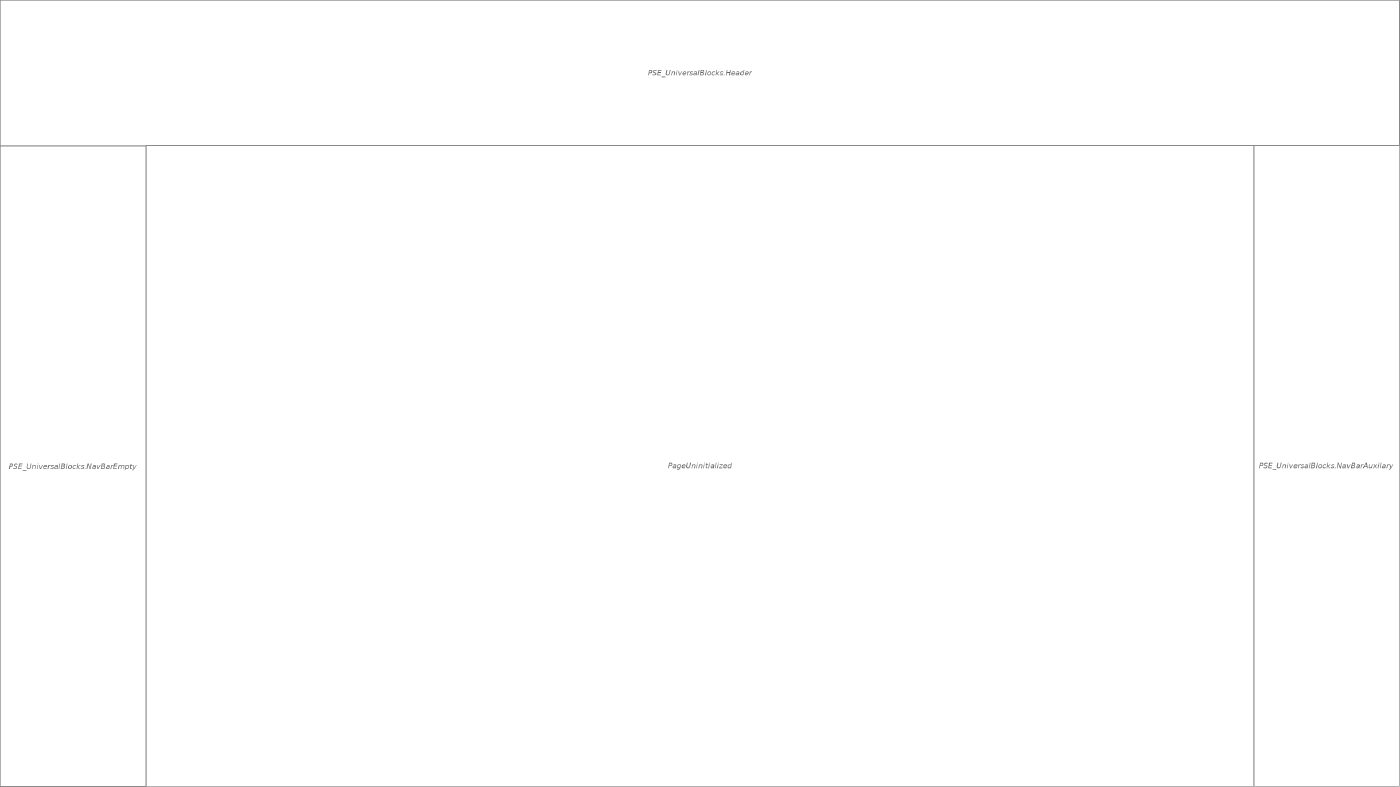
VISUALIZATION ShellMainVisu  // 1920x1080
    Frame (0,0 1920x200)
        shows PSE_UniversalBlocks.Header(sMachineName := PRG_VisuControl.fbVisuControl.sMachineName, sSoftwareVersion := PRG_VisuControl.fbVisuControl.sSoftwareVersion, eMachineState := PRG_MachineControl.fbMachineControler.State, sCurrentRecipe := PRG_VisuControl.fbVisuControl.sCurrentRecipe, sCurrentUser := PRG_VisuControl.fbVisuControl.sCurrentUser, iActiveCriticals := PRG_VisuControl.fbVisuControl.iActiveCriticals, iActvieErrors := PRG_VisuControl.fbVisuControl.iActvieErrors, iActiveWarrnings := PRG_VisuControl.fbVisuControl.iActiveWarrnings, sCurrentDate := PRG_VisuControl.fbVisuControl.sCurrentDate, sCurrentTime := PRG_VisuControl.fbVisuControl.sCurrentTime)
    Frame (0,200 200x880), frame switch variable: PRG_VisuControl.fbVisuControl.eCurrentNavigation
        shows PSE_UniversalBlocks.NavBarEmpty()
        shows PSE_UniversalBlocks.NavBarUninitialized(btnInitialize := PRG_VisuControl.fbVisuControl.btnInit)
        shows PSE_UniversalBlocks.NavBarInitializing(btnAbort := PRG_VisuControl.fbVisuControl.btnAbort)
        shows PSE_UniversalBlocks.NavBarAuto(btnStart := PRG_VisuControl.fbVisuControl.btnStart, btnStop := PRG_VisuControl.fbVisuControl.btnStop, btnManualMode := PRG_VisuControl.fbVisuControl.btnManual, btnAbort := PRG_VisuControl.fbVisuControl.btnAbort, btnReset := PRG_VisuControl.fbVisuControl.btnReset, bVisStart := PRG_VisuControl.fbVisuControl.bStartDisable, bVisStop := PRG_VisuControl.fbVisuControl.bStopDisable)
        shows PSE_UniversalBlocks.NavBarManual(btnAutoMode := PRG_VisuControl.fbVisuControl.btnAuto, btnCylinders := PRG_VisuControl.fbVisuControl.btnManualCylinder, btnMotors := PRG_VisuControl.fbVisuControl.btnManualAxis, btnSafety := PRG_VisuControl.fbVisuControl.btnManualSafety, btnInputs := PRG_VisuControl.fbVisuControl.btnManualInputs, btnOutputs := PRG_VisuControl.fbVisuControl.btnManualOutputs, btnOthers := PRG_VisuControl.fbVisuControl.btnManualOthers, btnAbort := PRG_VisuControl.fbVisuControl.btnAbort, btnRobots := PRG_VisuControl.fbVisuControl.btnManualRobots)
        shows PSE_UniversalBlocks.NavBarUtilities(btnBack := PRG_VisuControl.fbVisuControl.btnBack)
        shows PSE_UniversalBlocks.NavBarManual(btnAutoMode := PRG_Visu_Control.fbVisuControl.btnAuto, btnCylinders := PRG_Visu_Control.fbVisuControl.btnManualCylinder, btnMotors := PRG_Visu_Control.fbVisuControl.btnManualAxis, btnSafety := PRG_Visu_Control.fbVisuControl.btnManualSafety, btnInputs := PRG_Visu_Control.fbVisuControl.btnManualInputs, btnOutputs := PRG_Visu_Control.fbVisuControl.btnManualOutputs, btnOthers := PRG_Visu_Control.fbVisuControl.btnManualOthers, btnAbort := PRG_Visu_Control.fbVisuControl.btnAbort)
        shows PSE_UniversalBlocks.NavBarUtilities()
        shows PSE_UniversalBlocks.NavBarManual()
        shows PSE_UniversalBlocks.NavBarAuxilary(btnAlarms := PRG_Visu_Control.fbVisuControl.btnAlarms, btnRecipes := PRG_Visu_Control.fbVisuControl.btnRecipes, btnLights := PRG_Visu_Control.fbVisuControl.btnLights, sCloseHMIFileName := PRG_Visu_Control.fbVisuControl.sCloseHMIFileName, sCloseHMIParameters := PRG_Visu_Control.fbVisuControl.sCloseHMIParameters, bVisNotInit := PRG_Visu_Control.fbVisuControl.bVisNotInit, bVisHmiCLose := PRG_Visu_Control.fbVisuControl.bVisHmiClose, bVisLogIn := PRG_Visu_Control.fbVisuControl.bVisLogIn, bVisLogOut := PRG_Visu_Control.fbVisuControl.bVisLogOut)
        p2191133907: PRG_FB_Visu_Test.fbVisuControl.btnTest
        p3449907010: PRG_FB_Visu_Test.fbVisuControl.btnProcess
        p1834510317: PRG_FB_Visu_Test.fbVisuControl.btnTest
        p272088775: PRG_FB_Visu_Test.fbVisuControl.btnProcess
        p1969354770: PRG_FB_Visu_Test.fbVisuControl.btnAbort
        p1714963132: PRG_FB_Visu_Test.fbVisuControl.btnPushersScreenEntry
        p2303688632: PRG_FB_Visu_Test.fbVisuControl.btnStartAuto
        p3820184681: PRG_FB_Visu_Test.fbVisuControl.btnStop
        p1769496127: PRG_FB_Visu_Test.fbVisuControl.btnStepMode
        p2661042519: PRG_FB_Visu_Test.fbVisuControl.btnManual
        p976602031: PRG_VisuControl.fbVisuControl.btnBack
        p864465659: PRG_Visu_Control.fbVisuControl.ifUniversalMachineLink
        p1643820539: PRG_Visu_Control.fbVisuControl.btnStart
        p4004320302: PRG_Visu_Control.fbVisuControl.btnStop
        p3440189619: PRG_Visu_Control.fbVisuControl.btnManual
        p2317368076: PRG_Visu_Control.fbVisuControl.bVisStart
        p974511339: PRG_Visu_Control.fbVisuControl.bVisStop
        p3194361968: PRG_VisuControl.fbVisuControl.btnAuto
        p3852855334: PRG_VisuControl.fbVisuControl.btnManualCylinder
        p2703927093: PRG_VisuControl.fbVisuControl.btnManualAxis
        p1724788453: PRG_VisuControl.fbVisuControl.btnManualSafety
        p3478313700: PRG_VisuControl.fbVisuControl.btnManualInputs
        p985323216: PRG_VisuControl.fbVisuControl.btnManualOutputs
        p3968519516: PRG_VisuControl.fbVisuControl.btnManualOthers
        p3317205904: PRG_VisuControl.fbVisuControl.btnAbort
        p1887615166: PRG_VisuControl.fbVisuControl.btnManualRobots
    Frame (1719,199 200x880)
        shows PSE_UniversalBlocks.NavBarAuxilary(btnAlarms := PRG_VisuControl.fbVisuControl.btnAlarms, btnRecipes := PRG_VisuControl.fbVisuControl.btnRecipes, btnDoorLock := PRG_VisuControl.fbVisuControl.btnLights, btnLogIn := PRG_VisuControl.fbVisuControl.btnLogIn, btnLogOut := PRG_VisuControl.fbVisuControl.btnLogOut, btnHmiClose := PRG_VisuControl.fbVisuControl.btnHmiClose, sCloseHMIFileName := PRG_VisuControl.fbVisuControl.sCloseHMIFileName, sCloseHMIParameters := PRG_VisuControl.fbVisuControl.sCloseHMIParameters, bVisNotInit := PRG_VisuControl.fbVisuControl.bVisNotInit, bVisHmiCLose := PRG_VisuControl.fbVisuControl.bVisHmiClose, bVisLogIn := PRG_VisuControl.fbVisuControl.bVisLogIn, bVisLogOut := PRG_VisuControl.fbVisuControl.bVisLogOut, bDoorLockDisabled := PRG_VisuControl.fbVisuControl.btnLights, bDoorLockInvisible := PRG_VisuControl.fbVisuControl.btnLights)
        p1814871890: PRG_VisuControl.fbVisuControl.btnLights
        p741195761: PRG_VisuControl.fbVisuControl.btnAlarms
        p1428156847: PRG_VisuControl.fbVisuControl.btnRecipes
        p3449825089: PRG_VisuControl.fbVisuControl.btnLights
        p2958599044: PRG_VisuControl.fbVisuControl.btnLogIn
        p3266638362: PRG_VisuControl.fbVisuControl.btnLogOut
        p1254146404: PRG_VisuControl.fbVisuControl.btnHmiClose
        p2737420936: PRG_VisuControl.fbVisuControl.sCloseHMIFileName
        p411918085: PRG_VisuControl.fbVisuControl.sCloseHMIParameters
        p3390077939: PRG_VisuControl.fbVisuControl.bVisNotInit
        p777737485: PRG_VisuControl.fbVisuControl.bVisHmiClose
        p2994140705: PRG_VisuControl.fbVisuControl.bVisLogIn
        p1678412584: PRG_VisuControl.fbVisuControl.bVisLogOut
        p3450300924: PRG_VisuControl.fbVisuControl.btnLights
        p3107320333: PRG_VisuControl.fbVisuControl.btnLights
    Frame (200,199 1520x880), frame switch variable: PRG_VisuControl.fbVisuControl.eCurrentScreen
        shows PageUninitialized()
        shows PageInitializing(iProgressBar := PRG_VisuControl.fbVisuControl.iInitProgressBar)
        shows PSE_UniversalBlocks.PageReadyInitialized()
        shows PageAuto()
        shows PSE_UniversalBlocks.PageSwitchMode()
        shows PSE_UniversalBlocks.PageManualCylinders(btnPrevious := PRG_VisuControl.fbVisuControl.btnPrevious, btnNext := PRG_VisuControl.fbVisuControl.btnNext, bPreviousInvisible := PRG_VisuControl.fbVisuControl.bPreviousInvisible, bNextInvisible := PRG_VisuControl.fbVisuControl.bNextInvisible, stCylinderEmpty := PRG_VisuControl.fbVisuControl.arrCylinderFrameEmpty[PRG_VisuControl.fbVisuControl.iSelectedCylinderPageIndex], stCyliner := PRG_VisuControl.fbVisuControl.arrCylinderFrame[PRG_VisuControl.fbVisuControl.iSelectedCylinderPageIndex], iCylinderSelectedPageIndex := PRG_VisuControl.fbVisuControl.iSelectedCylinderPageIndex, iCylinderTotalPageIndex := PRG_VisuControl.fbVisuControl.iCylinderPageIndex)
        shows PSE_UniversalBlocks.PageManualAxis(btnPrevious := PRG_VisuControl.fbVisuControl.btnPrevious, btnNext := PRG_VisuControl.fbVisuControl.btnNext, bPreviousInvisible := PRG_VisuControl.fbVisuControl.bPreviousInvisible, bNextInvisible := PRG_VisuControl.fbVisuControl.bNextInvisible, stAxisEmpty := PRG_VisuControl.fbVisuControl.arrAxisFrameEmpty[PRG_VisuControl.fbVisuControl.iSelectedAxisPageIndex], stAxis := PRG_VisuControl.fbVisuControl.arrAxisFrame[PRG_VisuControl.fbVisuControl.iSelectedAxisPageIndex], iAxisSelectedPageIndex := PRG_VisuControl.fbVisuControl.iSelectedAxisPageIndex, iAxisTotalPageIndex := PRG_VisuControl.fbVisuControl.iAxisPageIndex)
        shows PSE_UniversalBlocks.PageManualInputs(btnPrevious := PRG_VisuControl.fbVisuControl.btnPrevious, btnNext := PRG_VisuControl.fbVisuControl.btnNext, bPreviousInvisible := PRG_VisuControl.fbVisuControl.bPreviousInvisible, bNextInvisible := PRG_VisuControl.fbVisuControl.bNextInvisible, stDigitalInputEmpty := PRG_VisuControl.fbVisuControl.arrInputFrameEmpty[PRG_VisuControl.fbVisuControl.iSelectedInputPageIndex], stDigitalInputData := PRG_VisuControl.fbVisuControl.arrInputFrame[PRG_VisuControl.fbVisuControl.iSelectedInputPageIndex], iInputSelectedPageIndex := PRG_VisuControl.fbVisuControl.iSelectedInputPageIndex, iInputTotalPageIndex := PRG_VisuControl.fbVisuControl.iInputPageIndex)
        shows PSE_UniversalBlocks.PageManualOutputs(btnPrevious := PRG_VisuControl.fbVisuControl.btnPrevious, btnNext := PRG_VisuControl.fbVisuControl.btnNext, bPreviousInvisible := PRG_VisuControl.fbVisuControl.bPreviousInvisible, bNextInvisible := PRG_VisuControl.fbVisuControl.bNextInvisible, stDigitalOutputEmpty := PRG_VisuControl.fbVisuControl.arrOutputFrameEmpty[PRG_VisuControl.fbVisuControl.iSelectedOutputPageIndex], stDigitalOutputData := PRG_VisuControl.fbVisuControl.arrOutputFrame[PRG_VisuControl.fbVisuControl.iSelectedOutputPageIndex], iOutputSelectedPageIndex := PRG_VisuControl.fbVisuControl.iSelectedOutputPageIndex, iOutputTotalPageIndex := PRG_VisuControl.fbVisuControl.iOutputPageIndex)
        shows PSE_UniversalBlocks.PageManualRobots(btnPrevious := PRG_VisuControl.fbVisuControl.btnPrevious, btnNext := PRG_VisuControl.fbVisuControl.btnNext, bPreviousInvisible := PRG_VisuControl.fbVisuControl.bPreviousInvisible, bNextInvisible := PRG_VisuControl.fbVisuControl.bNextInvisible, stRobotEmpty := PRG_VisuControl.fbVisuControl.arrRobotFrameEmpty[PRG_VisuControl.fbVisuControl.iSelectedRobotPageIndex], stRobot := PRG_VisuControl.fbVisuControl.arrRobotFrame[PRG_VisuControl.fbVisuControl.iSelectedRobotPageIndex], iRobotSelectedPageIndex := PRG_VisuControl.fbVisuControl.iSelectedRobotPageIndex, iRobotTotalPageIndex := PRG_VisuControl.fbVisuControl.iRobotPageIndex)
        shows PageManualOther()
        shows PSE_UniversalBlocks.PageAlarms(btnClearAllAlarms := PRG_VisuControl.fbVisuControl.btnClearAll, btnExportEvents := PRG_VisuControl.fbVisuControl.btnExport, iActiveAlarms := PRG_VisuControl.fbVisuControl.iActiveAlarms, iActiveCritical := PRG_VisuControl.fbVisuControl.iActiveCriticals, iActiveErrors := PRG_VisuControl.fbVisuControl.iActvieErrors, iActiveWarrnings := PRG_VisuControl.fbVisuControl.iActiveWarrnings, arrEvents := PRG_AlarmControl.fbAlarmControler.EventsTable, arrAlarms := PRG_AlarmControl.fbAlarmControler.AlarmsTable)
        shows PSE_UniversalBlocks.PageRecipesManager(btnCreate := PRG_VisuControl.fbVisuControl.btnCreate, btnSelect := PRG_VisuControl.fbVisuControl.btnSelect, btnLoad := PRG_VisuControl.fbVisuControl.btnLoad, btnRead := PRG_VisuControl.fbVisuControl.btnRead, btnReload := PRG_VisuControl.fbVisuControl.btnReload, btnBackup := PRG_VisuControl.fbVisuControl.btnBackup, btnRestore := PRG_VisuControl.fbVisuControl.btnRestore, btnRecipeNext := PRG_VisuControl.fbVisuControl.btnRecipeNext, btnRecipePrevious := PRG_VisuControl.fbVisuControl.btnRecipePrevious, btnRemove := PRG_VisuControl.fbVisuControl.btnRemove, btnReloadExternal := PRG_VisuControl.fbVisuControl.btnReloadExternal, bReloadInvisible := PRG_VisuControl.fbVisuControl.bReloadInvisible, bRecipeNextInvisible := PRG_VisuControl.fbVisuControl.bRecipeNextInvisible, bRecipePreviousInvisible := PRG_VisuControl.fbVisuControl.bRecipePreviousInvisible, bRecipeCreateInvisible := PRG_VisuControl.fbVisuControl.bRecipeCreateInvisible, bRecipeBackupRestoreInvisible := PRG_VisuControl.fbVisuControl.bRecipeBackupRestoreInvisible, bNoRecipeSelected := PRG_VisuControl.fbVisuControl.bNoRecipeSelected, bRecipeCreateDisabled := PRG_VisuControl.fbVisuControl.bCreateRecipeDisabled, bRecipeBackupRestoreDisabled := PRG_VisuControl.fbVisuControl.bBackupRestoreDisabled, bError := PRG_VisuControl.fbVisuControl.bRecipesManagerError, eRecipesManagerReturns := PRG_VisuControl.fbVisuControl.eRecipesManagerReturns, eReacipeManagerState := PRG_VisuControl.fbVisuControl.eRecipesManagerState, iSelectedRecipe := PRG_VisuControl.fbVisuControl.iSelectedRecipe, sSelectedRecipe := PRG_VisuControl.fbVisuControl.sSelectedRecipe, sNewRecipeName := PRG_VisuControl.fbVisuControl.sNewRecipeName, sRestoreBackupPath := PRG_VisuControl.fbVisuControl.sBackupStoragePath, sRestoreBackupRecipeName := PRG_VisuControl.fbVisuControl.sBackupRestoreRecipeName, arrRecipeNames := PRG_VisuControl.fbVisuControl.arrRecipesNames, arrRecipeParameterFrameEmpty := PRG_VisuControl.fbVisuControl.arrRecipeParameterFrameEmpty[PRG_VisuControl.fbVisuControl.iSelectedRecipeParameterPageIndex], arrRecipeParameterFrameData := PRG_VisuControl.fbVisuControl.arrRecipeParameterFrameData[PRG_VisuControl.fbVisuControl.iSelectedRecipeParameterPageIndex], arrRecipeParameterFrameType := PRG_VisuControl.fbVisuControl.arrRecipeParameterFrameType[PRG_VisuControl.fbVisuControl.iSelectedRecipeParameterPageIndex], iRecipeSelectedPageIndex := PRG_VisuControl.fbVisuControl.iSelectedRecipeParameterPageIndex, iRecipeTotalPageIndex := PRG_VisuControl.fbVisuControl.iRecipeParameterPageIndex)
        shows PSE_UniversalBlocks.PageReset()
        shows PSE_UniversalBlocks.PageAborting()
        shows PSE_UniversalBlocks.PageAborting()
        shows PSE_UniversalBlocks.PageAborting()
        shows PSE_UniversalBlocks.PageAborting()
        p326653322: PRG_FB_Visu_Test.fbVisuControl.arrInputFrameExist[PRG_FB_Visu_Test.fbVisuControl.iSelectedInputPageIndex]
        p3157872260: PRG_FB_Visu_Test.fbVisuControl.arrInputFrame[PRG_FB_Visu_Test.fbVisuControl.iSelectedInputPageIndex]
        p3240474043: PRG_FB_Visu_Test.fbVisuControl.arrOutputFrameExist[PRG_FB_Visu_Test.fbVisuControl.iSelectedOutputPageIndex]
        p379669430: PRG_FB_Visu_Test.fbVisuControl.arrMotorFrame[PRG_FB_Visu_Test.fbVisuControl.iSelectedMotorPageIndex]
        p4218841056: PRG_FB_Visu_Test.fbVisuControl.arrMotorFrameExist[PRG_FB_Visu_Test.fbVisuControl.iSelectedMotorPageIndex]
        p3990153529: PRG_FB_Visu_Test.fbVisuControl.arrSafeOutputFrameExist[0]
        p3298724636: PRG_FB_Visu_Test.fbVisuControl.arrSafeOutputFrame[0]
        p4027064500: PRG_FB_Visu_Test.fbVisuControl.arrSafeInputFrameExist[0]
        p2940690956: PRG_FB_Visu_Test.fbVisuControl.arrSafeInputFrame[0]
        p1128973015: PRG_FB_Visu_Test.fbVisuControl.arrCylinderFrameExist[PRG_FB_Visu_Test.fbVisuControl.iSelectedCylinderPageIndex]
        p4042523238: PRG_FB_Visu_Test.fbVisuControl.arrAxisFrameExist[PRG_FB_Visu_Test.fbVisuControl.iSelectedAxisPageIndex]
        p4096565854: PRG_FB_Visu_Test.fbVisuControl.arrSafeOutputFrameExist[0]
        p1357094282: PRG_VisuControl.fbVisuControl.arrSafeOutputFrame[PRG_VisuControl.fbVisuControl.iSelectedSafeOutputPageIndex]
        p1685403170: PRG_FB_Visu_Test.fbVisuControl.arrSafeInputFrameExist[0]
        p3060428933: PRG_VisuControl.fbVisuControl.arrSafeInputFrame[PRG_VisuControl.fbVisuControl.iSelectedSafeInputPageIndex]
        p3637127434: PRG_FB_Visu_Test.fbVisuControl.arrInputFrameExist[PRG_FB_Visu_Test.fbVisuControl.iSelectedInputPageIndex]
        p565568266: PRG_VisuControl.fbVisuControl.arrSafeInputFrameEmpty[PRG_VisuControl.fbVisuControl.iSelectedSafeInputPageIndex]
        p2985064310: PRG_VisuControl.fbVisuControl.arrSafeOutputFrameEmpty[PRG_VisuControl.fbVisuControl.iSelectedSafeOutputPageIndex]
        p529959495: PRG_VisuControl.fbVisuControl.arrOutputFrameEmpty[PRG_VisuControl.fbVisuControl.iSelectedOutputPageIndex]
        p4218742370: PRG_VisuControl.fbVisuControl.arrOutputFrame[PRG_VisuControl.fbVisuControl.iSelectedOutputPageIndex]
        p2658029867: PRG_Visu_Control.fbVisuControl.bCreateRecipeDisabled
        p1710962933: PRG_Visu_Control.fbVisuControl.bBackupRestoreDisabled
        p1441065260: PRG_Visu_Control.fbVisuControl.btnNext
        p465346691: PRG_Visu_Control.fbVisuControl.btnPrevious
        p2280985692: PRG_Visu_Control.fbVisuControl.arrRecipeParameterFrame[PRG_Visu_Control.fbVisuControl.iSelectedRecipeParameterPageIndex]
        p3467742188: PRG_Visu_Control.fbVisuControl.btnCreate
        p177570263: PRG_Visu_Control.fbVisuControl.btnSelect
        p840799744: PRG_Visu_Control.fbVisuControl.btnLoad
        p2404135802: PRG_Visu_Control.fbVisuControl.btnRead
        p3823084866: PRG_Visu_Control.fbVisuControl.btnReload
        p2123872955: PRG_Visu_Control.fbVisuControl.btnBackup
        p973735221: PRG_Visu_Control.fbVisuControl.btnRecipeNext
        p1287159425: PRG_Visu_Control.fbVisuControl.btnRecipePrevious
        p71683411: PRG_Visu_Control.fbVisuControl.btnRestore
        p1185437942: PRG_Visu_Control.fbVisuControl.bReloadInvisible
        p68049249: PRG_Visu_Control.fbVisuControl.bRecipeNextInvisible
        p2844414756: PRG_Visu_Control.fbVisuControl.bPreviousInvisible
        p2659393543: PRG_Visu_Control.fbVisuControl.bRecipeCreateInvisible
        p666764911: PRG_Visu_Control.fbVisuControl.bRecipeBackupRestoreInvisible
        p583444731: PRG_Visu_Control.fbVisuControl.bBackupRestoreDisabled
        p2033502605: PRG_Visu_Control.fbVisuControl.bCreateRecipeDisabled
        p3864355643: PRG_Visu_Control.fbVisuControl.bRecipesManagerError
        p3524053556: PRG_Visu_Control.fbVisuControl.eRecipesManagerReturns
        p1087861978: PRG_Visu_Control.fbVisuControl.eRecipesManagerState
        p3317198642: PRG_Visu_Control.fbVisuControl.iSelectedRecipe
        p3872755051: PRG_Visu_Control.fbVisuControl.sSelectedRecipe
        p1117055398: PRG_Visu_Control.fbVisuControl.sCreateRecipe
        p2291178852: PRG_Visu_Control.fbVisuControl.sRestoreBackupPath
        p1581747850: PRG_Visu_Control.fbVisuControl.arrRecipesNames
        p2009918513: PRG_Visu_Control.fbVisuControl.arrRecipeParameterFrameEmpty[PRG_Visu_Control.fbVisuControl.iSelectedRecipeParameterPageIndex]
        p2090952880: PRG_Visu_Control.fbVisuControl.arrRecipeParameterFrameData[PRG_Visu_Control.fbVisuControl.iSelectedRecipeParameterPageIndex]
        p1569508602: PRG_Visu_Control.fbVisuControl.arrRecipeParameterFrameType[PRG_Visu_Control.fbVisuControl.iSelectedRecipeParameterPageIndex]
        p2215290544: PRG_Visu_Control.fbVisuControl.iSelectedRecipeParameterPageIndex
        p2243811169: PRG_Visu_Control.fbVisuControl.iRecipeParameterPageIndex
        p3296751590: PRG_Visu_Control.fbVisuControl.btnPrevious
        p450871899: PRG_Visu_Control.fbVisuControl.btnNext
        p3964086746: PRG_Visu_Control.fbVisuControl.bPreviousInvisible
        p2742356004: PRG_Visu_Control.fbVisuControl.bNextInvisible
        p2765918274: PRG_Visu_Control.fbVisuControl.arrOutputFrameEmpty[PRG_Visu_Control.fbVisuControl.iSelectedOutputPageIndex]
        p3123306711: PRG_Visu_Control.fbVisuControl.arrOutputFrame[PRG_Visu_Control.fbVisuControl.iSelectedOutputPageIndex]
        p324713663: PRG_Visu_Control.fbVisuControl.iSelectedOutputPageIndex
        p2546208209: PRG_Visu_Control.fbVisuControl.iOutputPageIndex
        p636398411: PRG_VisuControl.fbVisuControl.btnPrevious
        p506073702: PRG_VisuControl.fbVisuControl.btnNext
        p142813351: PRG_VisuControl.fbVisuControl.bPreviousInvisible
        p2001311971: PRG_VisuControl.fbVisuControl.bNextInvisible
        p3845085143: PRG_Visu_Control.fbVisuControl.arrInputFrameEmpty[PRG_Visu_Control.fbVisuControl.iSelectedInputPageIndex]
        p1301550460: PRG_Visu_Control.fbVisuControl.arrInputFrame[PRG_Visu_Control.fbVisuControl.iSelectedInputPageIndex]
        p2725722896: PRG_Visu_Control.fbVisuControl.iSelectedInputPageIndex
        p2433681071: PRG_Visu_Control.fbVisuControl.iInputPageIndex
        p2125431502: PRG_Visu_Control.fbVisuControl.arrAxisFrameEmpty[PRG_Visu_Control.fbVisuControl.iSelectedAxisPageIndex]
        p2776987204: PRG_Visu_Control.fbVisuControl.arrAxisFrame[PRG_Visu_Control.fbVisuControl.iSelectedAxisPageIndex]
        p1577962829: PRG_Visu_Control.fbVisuControl.iSelectedAxisPageIndex
        p965901929: PRG_Visu_Control.fbVisuControl.iAxisPageIndex
        p267916118: PRG_Visu_Control.fbVisuControl.arrCylinderFrameEmpty[PRG_Visu_Control.fbVisuControl.iSelectedCylinderPageIndex]
        p3390772661: PRG_Visu_Control.fbVisuControl.arrCylinderFrame[PRG_Visu_Control.fbVisuControl.iSelectedCylinderPageIndex]
        p3333323384: PRG_Visu_Control.fbVisuControl.iSelectedCylinderPageIndex
        p3966342745: PRG_Visu_Control.fbVisuControl.iSelectedCylinderPageIndex
        p1075172589: PRG_Visu_Control.fbVisuControl.arrSafeInputFrame[0]
        p1646949828: PRG_Visu_Control.fbVisuControl.arrSafeInputFrameEmpty[0]
        p326896452: PRG_Visu_Control.fbVisuControl.arrSafeOutputFrame[0]
        p3446867799: PRG_Visu_Control.fbVisuControl.arrSafeOutputFrameEmpty[0]
        p3485161619: PRG_Visu_Control.fbVisuControl.iSafeOutputPageIndex
        p1731338485: PRG_Visu_Control.fbVisuControl.iSelectedSafeOutputPageIndex
        p1853071612: PRG_Visu_Control.fbVisuControl.iSelectedSafeInputPageIndex
        p1803585147: PRG_Visu_Control.fbVisuControl.iSafeInputPageIndex
        p217787018: PRG_Visu_Control.fbVisuControl.bPreviousInvisibleOutput
        p3235470863: PRG_Visu_Control.fbVisuControl.bNextInvisibleOutput
        p1199213480: PRG_Visu_Control.fbVisuControl.bPreviousInvisibleInput
        p1769577244: PRG_Visu_Control.fbVisuControl.bNextInvisibleInput
        p3246196278: PRG_Visu_Control.fbVisuControl.btnPreviousOutput
        p858909533: PRG_Visu_Control.fbVisuControl.btnNextOutput
        p374383709: PRG_Visu_Control.fbVisuControl.btnPreviousInput
        p951943438: PRG_Visu_Control.fbVisuControl.btnNextInput
        p2527438113: PRG_VisuControl.fbVisuControl.sCreateRecipe
        p1815429779: PRG_VisuControl.fbVisuControl.btnNextInput
        p1439642259: PRG_VisuControl.fbVisuControl.btnPreviousInput
        p3185282151: PRG_VisuControl.fbVisuControl.btnNextOutput
        p3185735191: PRG_VisuControl.fbVisuControl.btnPreviousOutput
        p3051586396: PRG_VisuControl.fbVisuControl.bNextInvisibleInput
        p3398491442: PRG_VisuControl.fbVisuControl.bPreviousInvisibleInput
        p3067708807: PRG_VisuControl.fbVisuControl.bNextInvisibleOutput
        p481081990: PRG_VisuControl.fbVisuControl.bPreviousInvisibleOutput
        p3810990021: PRG_VisuControl.fbVisuControl.iSelectedSafeInputPageIndex
        p2077693559: PRG_VisuControl.fbVisuControl.iSafeInputPageIndex
        p951778378: PRG_VisuControl.fbVisuControl.iSelectedSafeOutputPageIndex
        p3323806504: PRG_VisuControl.fbVisuControl.iSafeOutputPageIndex
        p3876959044: PRG_VisuControl.fbVisuControl.iOutputPageIndex
        p1662035872: PRG_VisuControl.fbVisuControl.iSelectedOutputPageIndex
        p1553999255: PRG_VisuControl.fbVisuControl.iInputPageIndex
        p1892632301: PRG_VisuControl.fbVisuControl.iSelectedInputPageIndex
        p1878409780: PRG_VisuControl.fbVisuControl.arrInputFrame[PRG_VisuControl.fbVisuControl.iSelectedInputPageIndex]
        p2634742818: PRG_VisuControl.fbVisuControl.arrInputFrameEmpty[PRG_VisuControl.fbVisuControl.iSelectedInputPageIndex]
        p3710705917: PRG_VisuControl.fbVisuControl.btnPrevious
        p4273876321: PRG_VisuControl.fbVisuControl.bPreviousInvisible
        p3497865195: PRG_VisuControl.fbVisuControl.bNextInvisible
        p322200097: PRG_VisuControl.fbVisuControl.btnNext
        p1581373886: PRG_VisuControl.fbVisuControl.arrRobotFrameEmpty[PRG_VisuControl.fbVisuControl.iSelectedRobotPageIndex]
        p2920217236: PRG_VisuControl.fbVisuControl.arrRobotFrame[PRG_VisuControl.fbVisuControl.iSelectedRobotPageIndex]
        p1876974057: PRG_VisuControl.fbVisuControl.iSelectedRobotPageIndex
        p4225494810: PRG_VisuControl.fbVisuControl.iRobotPageIndex
        p1444084988: PRG_VisuControl.fbVisuControl.btnCreate
        p2453075655: PRG_VisuControl.fbVisuControl.btnSelect
        p3560201540: PRG_VisuControl.fbVisuControl.btnLoad
        p1768290366: PRG_VisuControl.fbVisuControl.btnRead
        p2071777874: PRG_VisuControl.fbVisuControl.btnReload
        p3862220203: PRG_VisuControl.fbVisuControl.btnBackup
        p426409536: PRG_VisuControl.fbVisuControl.btnRestore
        p1079236643: PRG_VisuControl.fbVisuControl.btnRecipeNext
        p1731374750: PRG_VisuControl.fbVisuControl.btnRecipePrevious
        p2015548748: PRG_VisuControl.fbVisuControl.bReloadInvisible
        p2669744678: PRG_VisuControl.fbVisuControl.bRecipeNextInvisible
        p2789679904: PRG_VisuControl.fbVisuControl.bRecipePreviousInvisible
        p3233151730: PRG_VisuControl.fbVisuControl.bRecipeCreateInvisible
        p2817399279: PRG_VisuControl.fbVisuControl.bRecipeBackupRestoreInvisible
        p2434216693: PRG_VisuControl.fbVisuControl.bCreateRecipeDisabled
        p398386030: PRG_VisuControl.fbVisuControl.bBackupRestoreDisabled
        p2898404980: PRG_VisuControl.fbVisuControl.bRecipesManagerError
        p2352615617: PRG_VisuControl.fbVisuControl.eRecipesManagerReturns
        p3690479517: PRG_VisuControl.fbVisuControl.eRecipesManagerState
        p557977301: PRG_VisuControl.fbVisuControl.iSelectedRecipe
        p36695180: PRG_VisuControl.fbVisuControl.sSelectedRecipe
        p952972464: PRG_VisuControl.fbVisuControl.sNewRecipeName
        p95623745: PRG_VisuControl.fbVisuControl.sBackupStoragePath
        p2867421702: PRG_VisuControl.fbVisuControl.arrRecipesNames
        p1119135652: PRG_VisuControl.fbVisuControl.arrRecipeParameterFrameEmpty[PRG_VisuControl.fbVisuControl.iSelectedRecipeParameterPageIndex]
        p2973894552: PRG_VisuControl.fbVisuControl.arrRecipeParameterFrameData[PRG_VisuControl.fbVisuControl.iSelectedRecipeParameterPageIndex]
        p2423235538: PRG_VisuControl.fbVisuControl.arrRecipeParameterFrameType[PRG_VisuControl.fbVisuControl.iSelectedRecipeParameterPageIndex]
        p2345129652: PRG_VisuControl.fbVisuControl.iSelectedRecipeParameterPageIndex
        p1839082521: PRG_VisuControl.fbVisuControl.iRecipeParameterPageIndex
        p579474803: PRG_VisuControl.fbVisuControl.btnCreate
        p3870170952: PRG_VisuControl.fbVisuControl.btnSelect
        p921191997: PRG_VisuControl.fbVisuControl.btnLoad
        p2344215367: PRG_VisuControl.fbVisuControl.btnRead
        p266615773: PRG_VisuControl.fbVisuControl.btnReload
        p2460754980: PRG_VisuControl.fbVisuControl.btnBackup
        p1679390744: PRG_VisuControl.fbVisuControl.btnRestore
        p3182043222: PRG_VisuControl.fbVisuControl.btnRecipeNext
        p2255882253: PRG_VisuControl.fbVisuControl.btnRecipePrevious
        p3319589048: PRG_VisuControl.fbVisuControl.btnRemove
        p2581438414: PRG_VisuControl.fbVisuControl.btnReloadExternal
        p840719879: PRG_VisuControl.fbVisuControl.bReloadInvisible
        p3919088264: PRG_VisuControl.fbVisuControl.bRecipeNextInvisible
        p1955751334: PRG_VisuControl.fbVisuControl.bRecipePreviousInvisible
        p249890394: PRG_VisuControl.fbVisuControl.bRecipeCreateInvisible
        p528157562: PRG_VisuControl.fbVisuControl.bRecipeBackupRestoreInvisible
        p2688552560: PRG_VisuControl.fbVisuControl.bNoRecipeSelected
        p2685339010: PRG_VisuControl.fbVisuControl.bCreateRecipeDisabled
        p1057585497: PRG_VisuControl.fbVisuControl.bBackupRestoreDisabled
        p3366144957: PRG_VisuControl.fbVisuControl.bRecipesManagerError
        p1114303593: PRG_VisuControl.fbVisuControl.eRecipesManagerReturns
        p2906761011: PRG_VisuControl.fbVisuControl.eRecipesManagerState
        p3228304561: PRG_VisuControl.fbVisuControl.iSelectedRecipe
        p3808552680: PRG_VisuControl.fbVisuControl.sSelectedRecipe
        p2916107464: PRG_VisuControl.fbVisuControl.sNewRecipeName
        p1817484313: PRG_VisuControl.fbVisuControl.sBackupStoragePath
        p2298141503: PRG_VisuControl.fbVisuControl.sBackupRestoreRecipeName
        p2323324493: PRG_VisuControl.fbVisuControl.arrRecipesNames
        p1778597267: PRG_VisuControl.fbVisuControl.arrRecipeParameterFrameEmpty[PRG_VisuControl.fbVisuControl.iSelectedRecipeParameterPageIndex]
        p73445024: PRG_VisuControl.fbVisuControl.arrRecipeParameterFrameData[PRG_VisuControl.fbVisuControl.iSelectedRecipeParameterPageIndex]
        p625806058: PRG_VisuControl.fbVisuControl.arrRecipeParameterFrameType[PRG_VisuControl.fbVisuControl.iSelectedRecipeParameterPageIndex]
        p1494388786: PRG_VisuControl.fbVisuControl.iSelectedRecipeParameterPageIndex
        p1552292718: PRG_VisuControl.fbVisuControl.iRecipeParameterPageIndex
END_VISUALIZATION

(* stored: Version 1.1.0.1, ProductVersion 3.1.4024.9
   Visu ShellMainVisu: Id {bd474335-39c3-4210-8c65-27d4e58f2b2a} *)
